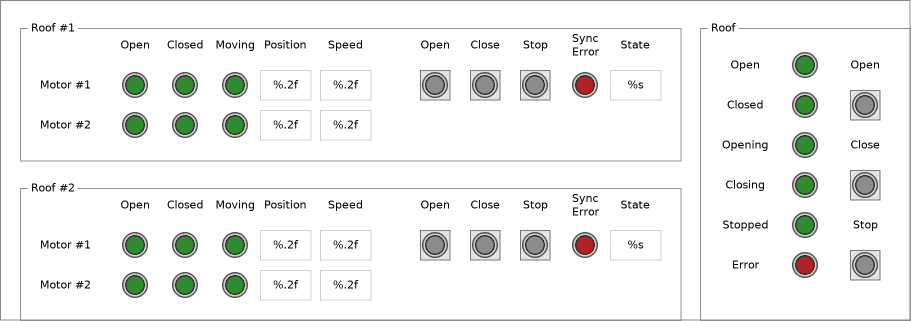
VISUALIZATION Visualization  // 911x321
    GroupBox (20,20 661x141), "Roof #1"
        Label (10,50 71x30), "Motor #1"
        Label (10,90 71x30), "Motor #2"
        Label (80,10 71x30), "Open"
        Label (130,10 71x30), "Closed"
        Lamp1 (100,50 30x30), variable: MAIN.RoofControl.roofs[1].motors[1].opened, style: Lamp-Lamp1-Green
        Lamp1 (150,50 30x30), variable: MAIN.RoofControl.roofs[1].motors[1].closed, style: Lamp-Lamp1-Green
        Lamp1 (100,90 30x30), variable: MAIN.RoofControl.roofs[1].motors[2].opened, style: Lamp-Lamp1-Green
        Lamp1 (150,90 30x30), variable: MAIN.RoofControl.roofs[1].motors[2].closed, style: Lamp-Lamp1-Green
        Label (180,10 71x30), "Moving"
        Lamp1 (200,50 30x30), variable: MAIN.RoofControl.roofs[1].motors[1].moving, style: Lamp-Lamp1-Green
        Lamp1 (200,90 30x30), variable: MAIN.RoofControl.roofs[1].motors[2].moving, style: Lamp-Lamp1-Green
        Label (230,10 71x30), "Position"
        Textfield (240,50 51x30), "%.2f", text variable: MAIN.RoofControl.roofs[1].motors[1].position, input disabled if: TRUE
        Textfield (240,90 51x30), "%.2f", text variable: MAIN.RoofControl.roofs[1].motors[2].position, input disabled if: TRUE
        Label (290,10 71x30), "Speed"
        Textfield (300,50 51x30), "%.2f", text variable: MAIN.RoofControl.roofs[1].motors[1].speed, input disabled if: TRUE
        Textfield (300,90 51x30), "%.2f", text variable: MAIN.RoofControl.roofs[1].motors[2].speed, input disabled if: TRUE
        Label (380,10 71x30), "Open"
        PushSwitch (400,50 30x30), variable: MAIN.RoofControl.open_roof1, behaviour: TAP, style: Switch-PushSwitch-Gray
        PushSwitch (450,50 30x30), variable: MAIN.RoofControl.close_roof1, behaviour: TAP, style: Switch-PushSwitch-Gray
        Label (430,10 71x30), "Close"
        Label (480,10 71x30), "Stop"
        PushSwitch (500,50 30x30), variable: MAIN.RoofControl.stop_roof1, behaviour: TAP, style: Switch-PushSwitch-Gray
        Lamp1 (550,50 30x30), variable: MAIN.RoofControl.roofs[1].sync_error, style: Lamp-Lamp1-Red
        Label (540,10 51x30), "Sync Error"
        Label (580,10 71x30), "State"
        Textfield (590,50 51x30), "%s", text variable: MAIN.RoofControl.roofs[1].state, input disabled if: TRUE
    GroupBox (20,180 661x141), "Roof #2"
        Label (10,50 71x30), "Motor #1"
        Label (10,90 71x30), "Motor #2"
        Label (80,10 71x30), "Open"
        Label (130,10 71x30), "Closed"
        Lamp1 (100,50 30x30), variable: MAIN.RoofControl.roofs[2].motors[1].opened, style: Lamp-Lamp1-Green
        Lamp1 (150,50 30x30), variable: MAIN.RoofControl.roofs[2].motors[1].closed, style: Lamp-Lamp1-Green
        Lamp1 (100,90 30x30), variable: MAIN.RoofControl.roofs[2].motors[2].opened, style: Lamp-Lamp1-Green
        Lamp1 (150,90 30x30), variable: MAIN.RoofControl.roofs[2].motors[2].closed, style: Lamp-Lamp1-Green
        Label (180,10 71x30), "Moving"
        Lamp1 (200,50 30x30), variable: MAIN.RoofControl.roofs[2].motors[1].moving, style: Lamp-Lamp1-Green
        Lamp1 (200,90 30x30), variable: MAIN.RoofControl.roofs[2].motors[2].moving, style: Lamp-Lamp1-Green
        Label (230,10 71x30), "Position"
        Textfield (240,50 51x30), "%.2f", text variable: MAIN.RoofControl.roofs[2].motors[1].position, input disabled if: TRUE
        Textfield (240,90 51x30), "%.2f", text variable: MAIN.RoofControl.roofs[2].motors[2].position, input disabled if: TRUE
        Label (290,10 71x30), "Speed"
        Textfield (300,50 51x30), "%.2f", text variable: MAIN.RoofControl.roofs[2].motors[1].speed, input disabled if: TRUE
        Textfield (300,90 51x30), "%.2f", text variable: MAIN.RoofControl.roofs[2].motors[2].speed, input disabled if: TRUE
        Label (380,10 71x30), "Open"
        PushSwitch (400,50 30x30), variable: MAIN.RoofControl.open_roof2, behaviour: TAP, style: Switch-PushSwitch-Gray
        PushSwitch (450,50 30x30), variable: MAIN.RoofControl.close_roof2, behaviour: TAP, style: Switch-PushSwitch-Gray
        Label (430,10 71x30), "Close"
        Label (480,10 71x30), "Stop"
        PushSwitch (500,50 30x30), variable: MAIN.RoofControl.stop_roof2, behaviour: TAP, style: Switch-PushSwitch-Gray
        Label (540,10 51x30), "Sync Error"
        Lamp1 (550,50 30x30), variable: MAIN.RoofControl.roofs[2].sync_error, style: Lamp-Lamp1-Red
        Label (580,10 71x30), "State"
        Textfield (590,50 51x30), "%s", text variable: MAIN.RoofControl.roofs[2].state, input disabled if: TRUE
    GroupBox (700,20 211x301), "Roof"
        Label (10,30 71x30), "Open"
        Label (10,70 71x30), "Closed"
        Lamp1 (90,30 30x30), variable: Main.RoofControl.opened, style: Lamp-Lamp1-Green
        Lamp1 (90,70 30x30), variable: Main.RoofControl.closed, style: Lamp-Lamp1-Green
        Label (10,110 71x30), "Opening"
        Lamp1 (90,110 30x30), variable: Main.RoofControl.opening, style: Lamp-Lamp1-Green
        Label (130,30 71x30), "Open"
        PushSwitch (150,70 30x30), variable: Main.open, behaviour: TAP, style: Switch-PushSwitch-Gray
        PushSwitch (150,150 30x30), variable: Main.close, behaviour: TAP, style: Switch-PushSwitch-Gray
        Label (130,110 71x30), "Close"
        Label (130,190 71x30), "Stop"
        PushSwitch (150,230 30x30), variable: Main.stop, behaviour: TAP, style: Switch-PushSwitch-Gray
        Label (10,150 71x30), "Closing"
        Lamp1 (90,150 30x30), variable: Main.RoofControl.closing, style: Lamp-Lamp1-Green
        Label (10,190 71x30), "Stopped"
        Lamp1 (90,190 30x30), variable: Main.RoofControl.stopped, style: Lamp-Lamp1-Green
        Label (10,230 71x30), "Error"
        Lamp1 (90,230 30x30), variable: Main.RoofControl.error, style: Lamp-Lamp1-Red
END_VISUALIZATION

(* stored: Version 1.1.0.1, ProductVersion 3.1.4024.13
   Visu Visualization: Id {e3a97d1b-e9a1-4ad0-8506-6ff5b42fdc2a} *)
